// LS Electric XG5000 project: counterTest
// PLC NewPLC
// module base 0 slot 0: 입출력 모듈:XBC-DR20S (DC 24V 입력 12점, 릴레이 출력 8점)

PROGRAM NewProgram (task: 스캔 프로그램)

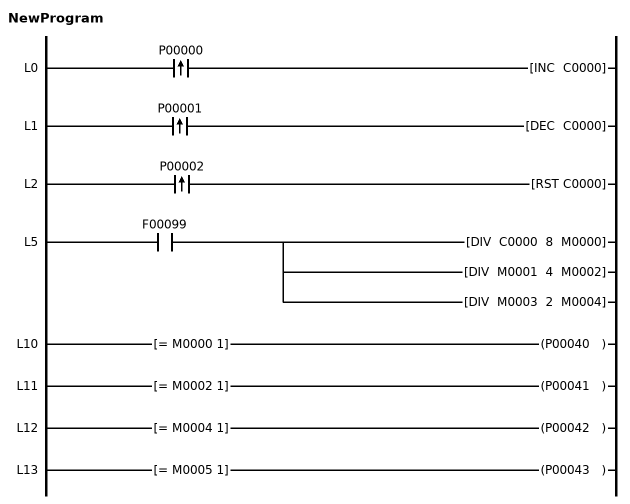
; L0
LOADP     P00000
INC       C0000
; L1
LOADP     P00001
DEC       C0000
; L2
LOADP     P00002
RST       C0000
; L5
LOAD      F00099
DIV       C0000 8 M0000
DIV       M0001 4 M0002
DIV       M0003 2 M0004
; L10
LOAD=     M0000 1
OUT       P00040
; L11
LOAD=     M0002 1
OUT       P00041
; L12
LOAD=     M0004 1
OUT       P00042
; L13
LOAD=     M0005 1
OUT       P00043